TYPE T_Comparison : E_COMPARISON; END_TYPE

(* stored: Version 1.1.0.1, ProductVersion 3.1.4024.4
   DUT T_Comparison: Id {4ba48f1e-17f2-075b-03e1-f6f1c9fe2c1d} *)
